PROGRAM P00_Task_Fast
VAR
END_VAR


Task_Fast_LH();
Task_Fast_TB();

END_PROGRAM

(* stored: Version 1.1.0.1, ProductVersion 3.1.4024.12
   POU P00_Task_Fast: Id {91a6d0eb-8720-440f-af9c-73126ec61acc}, SpecialFunc None *)
